// TIA Portal V16 export
// export: Created 2021-07-12T14:47:19.3566554Z, ExportSetting WithDefaults, DisplayName Totally Integrated Automation Portal, DisplayVersion V16, DisplayName TIA Portal Version Control Interface, DisplayVersion V16, DisplayName TIA Portal Openness, DisplayVersion V16, DisplayName STEP 7 Professional, DisplayVersion V16, DisplayName STEP 7 Safety, DisplayVersion V16, DisplayName WinCC Professional, DisplayVersion V16
TYPE "SimaHydTO_typeHMIConnection"
TITLE = SimaHydTO_typeHMIConnection
// HMI connection interface data block
// stored: IsFailsafeCompliant false
   STRUCT
      AxisData { S7_SetPoint := 'True'} : "SimaHydTO_typeHMIConnectionAxisData";
      AxisToData { S7_SetPoint := 'True'} : "SimaHydTO_typeHMIConnectionAxisToData";
      AxisSelector { S7_SetPoint := 'True'} : "SimaHydTO_typeHMIConnectionAxisSelector";
      BasicAxisControl { S7_SetPoint := 'True'} : "SimaHydTO_typeHMIConnectionBasicAxisControl";
      GetCharacteristics { S7_SetPoint := 'True'} : "SimaHydTO_typeHMIConnectionGetCharacteristicInterface";
      HmiData { S7_SetPoint := 'True'} : "SimaHydTO_typeHMIConnectionHmiData";
      VCharEditor { S7_SetPoint := 'True'} : "SimaHydTO_typeHMIConnectionVCharEditor";
      AdvancedAxisControl { S7_SetPoint := 'True'} : "SimaHydTO_typeHMIConnectionAdvancedAxisControl";
      ParameterSettings { S7_SetPoint := 'True'} : "SimaHydTO_typeHMIConnectionParameterSettings";
   END_STRUCT;
END_TYPE
